FUNCTION TryConvert_DATE_TO_DT : BOOL
VAR_INPUT
	in : DATE;
	out : REFERENCE TO DT;
END_VAR

IF in > DatatypeLimits.MAX_VALUE_OF_DATE_WHICH_CAN_BE_HELD_IN_A_DT THEN
	RETURN;
END_IF

out := DATE_TO_DT(in);
TryConvert_DATE_TO_DT := TRUE;

END_FUNCTION

(* stored: Version 1.1.0.1, ProductVersion 3.1.4024.12
   POU TryConvert_DATE_TO_DT: Id {0822ffca-fba3-4876-8078-009fd44eca05}, SpecialFunc None *)
